// TwinCAT 3 PLC project PLCSample
// ProgramVersion: 3.1.4020.4
// libraries:
//   Tc2_Standard, * (Beckhoff Automation GmbH)
//   Tc2_System, * (Beckhoff Automation GmbH)
//   Tc2_Utilities, * (Beckhoff Automation GmbH)
//   Tc3_Module, * (Beckhoff Automation GmbH)
// project tree:
//   / PlcTask.TcTTO
//   POUs/ FB_Engine.TcPOU, FB_NewEngine.TcPOU, MAIN.TcPOU
// real-time tasks:
//   TASK PlcTask: cycle T#10ms, priority 20, ADS port 350

CONFIGURATION PLCSample
    RESOURCE PLC ON TwinCAT3
        TASK PlcTask(INTERVAL := T#10ms, PRIORITY := 20);
        PROGRAM MAIN WITH PlcTask : MAIN;
    END_RESOURCE
END_CONFIGURATION

// ---- POUs/MAIN.TcPOU
PROGRAM MAIN
VAR
	fbNewEngine			: FB_NewEngine;	
END_VAR

fbNewEngine.Start(1, 7.5);

END_PROGRAM

// ---- POUs/FB_NewEngine.TcPOU
FUNCTION_BLOCK PUBLIC FB_NewEngine EXTENDS FB_Engine
VAR_INPUT
	nGear		:	INT := 2;
	fVelocity	:	LREAL := 8.0;
END_VAR
VAR
	gearInternal		:	INT;
END_VAR

{attribute 'monitoring' := 'variable'}
PROPERTY PUBLIC Gear : INT
GET
Gear := gearInternal;
END_GET
SET
gearInternal := Gear;
END_SET
END_PROPERTY

METHOD PUBLIC Start
VAR_INPUT
	nGear		:	INT := 2;
	fVelocity	:	LREAL := 8.0;
END_VAR
SUPER^.Start(nGear, fVelocity);
Gear := nGear;
END_METHOD

END_FUNCTION_BLOCK

// ---- POUs/FB_Engine.TcPOU
FUNCTION_BLOCK PUBLIC FB_Engine
VAR
	maxVelocityInternal		:	LREAL := 50.0;
	velocityInternal		:	LREAL;	
	temperatureInternal		:	INT;
END_VAR

{attribute 'monitoring' := 'variable'}
PROPERTY PUBLIC MaxVelocity : LREAL
GET
MaxVelocity := maxVelocityInternal;
END_GET
SET
maxVelocityInternal := MaxVelocity;
END_SET
END_PROPERTY

METHOD PUBLIC Start
VAR_INPUT
	nGear		:	INT := 2;
	fVelocity	:	LREAL := 8.0;
END_VAR
IF (fVelocity < MaxVelocity) THEN
	velocityInternal := fVelocity;
ELSE
	velocityInternal := MaxVelocity;
END_IF
END_METHOD

METHOD PUBLIC Stop
VAR_INPUT
END_VAR
velocityInternal := 0;
END_METHOD

{attribute 'monitoring' := 'variable'}
PROPERTY PUBLIC Temperature : INT
GET
Temperature := temperatureInternal;
END_GET
END_PROPERTY

{attribute 'monitoring' := 'variable'}
PROPERTY PUBLIC Velocity : LREAL
GET
Velocity := velocityInternal;
END_GET
END_PROPERTY

END_FUNCTION_BLOCK
